FUNCTION_BLOCK Test_DateAsString EXTENDS TUnitTestBase
VAR
END_VAR

METHOD  Execute
VAR_INST
    TimeStruct : TIMESTRUCT := (wDay := 23, wMonth := 12, wYear := 1945);
END_VAR
Assertion.AssertEquals_STRING(
    Expected := '23/12/1945',
    Actual   := F_DateAsString(TimeStruct),
    ObjectName := _TestName,
    VariableName  := 'F_DateAsString(TimeStruct)');


Test_Finished();
END_METHOD

END_FUNCTION_BLOCK

(* stored: Version 1.1.0.1, ProductVersion 3.1.4024.3
   POU Test_DateAsString: Id {01583d56-7c03-4d57-9b3f-326c17e75b06}, SpecialFunc None
   Method Execute: Id {8bb540d1-cab6-4c56-ac18-b399b5f13c6e} *)
